// TwinCAT 3 PLC project LoggingExample
// ProgramVersion: 3.1.4024.0
// libraries:
//   Core, 0.0.1.0 (Ziga)
//   Logging, 0.0.1.5 (Ziga)
//   Tc2_Standard, * (Beckhoff Automation GmbH)
//   Tc2_System, * (Beckhoff Automation GmbH)
//   Tc3_Module, * (Beckhoff Automation GmbH)
//   TcError, 0.2.2.0 (Roald87)
//   TcUnit, 1.3.1 (www.tcunit.org)
// project tree:
//   DUTs/ E_SimulationState.TcDUT
//   GVLs/ GVL.TcGVL
//   / PlcTask.TcTTO
//   POUs/ MAIN.TcPOU
//   POUs/Position observer/ FB_PositionObserver_LoggerWithDependencyInjection.TcPOU, FB_PositionObserver_OptionalLoggerWithDependencyInjection.TcPOU, FB_PositionSensorObserverBase.TcPOU
// real-time tasks:
//   TASK PlcTask: cycle T#10ms, priority 20, ADS port 350

CONFIGURATION LoggingExample
    RESOURCE PLC ON TwinCAT3
        TASK PlcTask(INTERVAL := T#10ms, PRIORITY := 20);
        PROGRAM MAIN WITH PlcTask : MAIN;
    END_RESOURCE
END_CONFIGURATION

// ---- DUTs/E_SimulationState.TcDUT
{attribute 'qualified_only'}
{attribute 'strict'}

// Adding this attribute allows to call TO_STRING(enumVariable), which will result in the name of the enum member
{attribute 'to_string'}

TYPE E_SimulationState :
(
	IDLE, 
	BOTTOM, 
	BOTTOM_FOR_10_SECONDS, 
	TOP, TOP_FOR_10_SECONDS 
):= IDLE;
END_TYPE

// ---- GVLs/GVL.TcGVL
{attribute 'qualified_only'}
VAR_GLOBAL
	Logger	: ZigaLibs_Logging.FB_Logger;
	ILogger	: ZigaLibs_Core.I_LoggerEx := Logger;
END_VAR

// ---- POUs/MAIN.TcPOU
PROGRAM MAIN
VAR
	// Instantiating the function block with logger via dependency injection.
	fbPositionObserver_WithLogger : 
		FB_PositionObserver_LoggerWithDependencyInjection(logger := GVL.Logger);
		
	// Instantiating the function block with provided optional logger via dependency injection.
	// For this to work, we need to provide the interface (pointer), instead of the instantiating function block.	
	fbPositionObserver_OptionalLogger_WithLogger : 
		FB_PositionObserver_OptionalLoggerWithDependencyInjection(logger := GVL.ILogger);
		
	// Instantiating the function block without logger via dependency injection.	
	fbPositionObserver_OptionalLogger_WithoutLogger : 
		FB_PositionObserver_OptionalLoggerWithDependencyInjection(logger := 0);
	
		
	eSimulationState			: E_SimulationState := E_SimulationState.IDLE;
	tonPositionTimer			: Tc2_Standard.TON();
	
	
	// Run the simulation
	SIMULATION_RUN				: BOOL;
	observer_simulationState	: ZigaLibs_Core.BoolEx := (variable := SIMULATION_RUN);
	sb							: ZigaLibs_Core.FB_StringBuilder;
	
	firstExecutionAndLoggerValid	: BOOL := TRUE;
END_VAR

VAR CONSTANT
	MY_TARGET_DEVICE_NET_ID 		: Tc2_System.T_AmsNetIdArr := [192,168,56,1,1,1]; // Empty = local
	MY_LOGGER_EXAMPLE_FILE_LOCATION	: Tc2_System.T_MaxString := 'C:\';
	MY_LOGGER_EXAMPLE_FILE_NAME		: Tc2_System.T_MaxString := 'ExampleLog';
END_VAR

// Configure logger
GVL.Logger.AmsAddress.netId := MY_TARGET_DEVICE_NET_ID; 
GVL.Logger.FileProperties.FileLocation := MY_LOGGER_EXAMPLE_FILE_LOCATION;
GVL.Logger.FileProperties.FileName := MY_LOGGER_EXAMPLE_FILE_NAME;

// Logger body still needs to be called
GVL.Logger();

IF GVL.Logger.Ready THEN
	IF firstExecutionAndLoggerValid THEN
		GVL.Logger.LogDefault('====================== FIRST PLC CYCLE EXECUTED ======================');
	END_IF
	firstExecutionAndLoggerValid := FALSE;
	
	// Start/stop simulation logging
	observer_simulationState();
	IF observer_simulationState.HasRisingEdge THEN
		GVL.Logger.LogDefault('====================== STARTING SIMULATION =============================');
		eSimulationState := E_SimulationState.IDLE;
	ELSIF observer_simulationState.HasFallingEdge THEN
		GVL.Logger.LogDefault('====================== STOPPING SIMULATION =============================');
	END_IF
END_IF

// Lets wait for logger to be ready, otherwise date time will be 1970
IF GVL.Logger.Ready AND SIMULATION_RUN THEN		
	// INFO: Check the "Set" implementation for the SimulationState property in MAIN. 
	// You can see state changes being logged in there as well.
	
	// Simulating the positions to generate logs
	CASE SimulationState OF
		E_SimulationState.IDLE:	
			fbPositionObserver_WithLogger.TopPositionSensor := FALSE;
			fbPositionObserver_WithLogger.BottomPositionSensor := FALSE;
			
			fbPositionObserver_OptionalLogger_WithLogger.TopPositionSensor := FALSE;
			fbPositionObserver_OptionalLogger_WithLogger.BottomPositionSensor := FALSE;
			
			fbPositionObserver_OptionalLogger_WithoutLogger.TopPositionSensor := FALSE;
			fbPositionObserver_OptionalLogger_WithoutLogger.BottomPositionSensor := FALSE;
			
			tonPositionTimer(IN := FALSE);
			SimulationState := E_SimulationState.BOTTOM;
			
		E_SimulationState.BOTTOM:
			fbPositionObserver_WithLogger.TopPositionSensor := FALSE;
			fbPositionObserver_WithLogger.BottomPositionSensor := TRUE;
			
			fbPositionObserver_OptionalLogger_WithLogger.TopPositionSensor := FALSE;
			fbPositionObserver_OptionalLogger_WithLogger.BottomPositionSensor := TRUE;
			
			fbPositionObserver_OptionalLogger_WithoutLogger.TopPositionSensor := FALSE;
			fbPositionObserver_OptionalLogger_WithoutLogger.BottomPositionSensor := TRUE;
	
			SimulationState := E_SimulationState.BOTTOM_FOR_10_SECONDS;
			
		E_SimulationState.BOTTOM_FOR_10_SECONDS:
		
			tonPositionTimer(IN := TRUE, PT := T#10S);
			IF tonPositionTimer.Q THEN
				tonPositionTimer(IN := FALSE);
				SimulationState := E_SimulationState.TOP;
			END_IF
			
		E_SimulationState.TOP:
			fbPositionObserver_WithLogger.TopPositionSensor := TRUE;
			fbPositionObserver_WithLogger.BottomPositionSensor := FALSE;
			
			fbPositionObserver_OptionalLogger_WithLogger.TopPositionSensor := TRUE;
			fbPositionObserver_OptionalLogger_WithLogger.BottomPositionSensor := FALSE;
			
			fbPositionObserver_OptionalLogger_WithoutLogger.TopPositionSensor := TRUE;
			fbPositionObserver_OptionalLogger_WithoutLogger.BottomPositionSensor := FALSE;
			
			SimulationState := E_SimulationState.TOP_FOR_10_SECONDS;
			
		E_SimulationState.TOP_FOR_10_SECONDS:
			tonPositionTimer(IN := TRUE, PT := T#10S);
			IF tonPositionTimer.Q THEN
				SimulationState := E_SimulationState.IDLE;
			END_IF
	END_CASE
END_IF


// Call the function blocks here, after simulation
fbPositionObserver_WithLogger();
fbPositionObserver_OptionalLogger_WithLogger();
fbPositionObserver_OptionalLogger_WithoutLogger();

// Gets or sets the simulation state
PROPERTY SimulationState : E_SimulationState
GET
SimulationState := eSimulationState;
END_GET
SET
// Check if value has changed, log the change as well.
IF SimulationState <> eSimulationState THEN
	GVL.Logger.LogDefault(sb.Reset()
		.AddString('========== SIMULATION STATE CHANGED FROM ')
		.AddWithDblQuotationMarks(TO_STRING(eSimulationState))
		.AddString(' TO ')
		.AddWithDblQuotationMarks(TO_STRING(eSimulationState))
		.AddString(' ========== ')
		.Create());
END_IF

eSimulationState := SimulationState;
END_SET
END_PROPERTY

END_PROGRAM

// ---- POUs/Position observer/FB_PositionObserver_LoggerWithDependencyInjection.TcPOU
// A function block with I_LoggerEX as required parameter passed trought FB_Init (dependency injection)
FUNCTION_BLOCK FB_PositionObserver_LoggerWithDependencyInjection EXTENDS FB_PositionSensorObserverBase

// Calling the base class body, FB_PositionSensorObserverBase. It assigns and calls the observers, triggers, ...
// If you want to change how the triggers behave, you could just not call SUPER and do your own implementaiton.
SUPER^();

// =======================================================================================
// ================================ WARNING ==============================================
// =======================================================================================
IF _bottoPositionObserver.HasRisingEdge THEN
	// Lets imagine the bottom position indicates a warning
	_logger.LogWarning(_sb.Reset()
		.AddString('Source: ')
		.AddWithDblQuotationMarks(THIS^.InstanceName)
		.AddString(' Bottom position reached.')
		.Create());
END_IF


// =======================================================================================
// ================================ ERROR ================================================
// =======================================================================================
// And after certain time, we need to trigger an error
IF _bottomPositionError.Q THEN
	_logger.LogError(_sb.Reset()
		.AddString('Source: ').AddWithDblQuotationMarks(THIS^.InstanceName)
		.AddString(' - bottom position has been active for too long!')
		.AddString('Maximum allowed duration is ').AddString(TO_STRING(MAXIMUM_DURATION_AT_BOTTOM_POSITION)).AddString('!')
		.Create());
END_IF

// =======================================================================================
// ================================ INFO =================================================
// =======================================================================================
IF _bottoPositionObserver.HasFallingEdge THEN
	_logger.LogInfo(_sb.Reset()
		.AddString('Source: ').AddWithDblQuotationMarks(THIS^.InstanceName)
		.AddString(' No longer at bottom position. ')
		.AddString('Bottom position was active for ')
		.Create());
END_IF

// =======================================================================================
// ================================ INFO =================================================
// =======================================================================================
IF _topPositionObserver.HasRisingEdge THEN
	_logger.LogInfo(_sb.Reset()
		.AddString('Source: ')
		.AddWithDblQuotationMarks(THIS^.InstanceName)
		.AddString(' Top position reached.')
		.Create());
END_IF

// =======================================================================================
// ================================ INFO =================================================
// =======================================================================================
IF _topPositionObserver.HasFallingEdge THEN
	_logger.LogInfo(_sb.Reset()
		.AddString('Source: ')
		.AddWithDblQuotationMarks(THIS^.InstanceName)
		.AddString(' No longer at top position.')
		.Create());
END_IF

METHOD FB_init : BOOL
VAR_INPUT
	bInitRetains : BOOL; // if TRUE, the retain variables are initialized (warm start / cold start)
	bInCopyCode : BOOL;  // if TRUE, the instance afterwards gets moved into the copy code (online change)
	logger	: ZigaLibs_Core.I_LoggerEx;
END_VAR
// Assign the internal interface to the one provided - interface is basically a pointer. Passing the address this way.
_logger := logger;
END_METHOD

END_FUNCTION_BLOCK

// ---- POUs/Position observer/FB_PositionSensorObserverBase.TcPOU
FUNCTION_BLOCK ABSTRACT FB_PositionSensorObserverBase EXTENDS ZigaLibs_Core.FB_HasInstanceName

VAR
	_topPositionObserver 	: ZigaLibs_Core.BoolEx;
	_topPositionError		: Tc2_Standard.R_TRIG;
	
	_bottoPositionObserver	: ZigaLibs_Core.BoolEx;
	_bottomPositionError	: Tc2_Standard.R_TRIG;
	
	_logger					: ZigaLibs_Core.I_LoggerEx;
	_sb						: ZigaLibs_Core.FB_StringBuilder;
END_VAR

VAR
	{attribute 'hide'}
	_topPositionSensor		: BOOL;
	{attribute 'hide'}
	_bottomPositionSensor	: BOOL;
END_VAR

VAR CONSTANT
	MAXIMUM_DURATION_AT_BOTTOM_POSITION : TIME := T#10S;
	MAXIMUM_DURATION_AT_TOP_POSITION 	: TIME := T#10S;
END_VAR

_topPositionObserver(variable := TopPositionSensor);
_bottoPositionObserver(variable := BottomPositionSensor);
_topPositionError(CLK := _topPositionObserver.HasBeenTrueForAtLeast(MAXIMUM_DURATION_AT_TOP_POSITION));
_bottomPositionError(CLK := _bottoPositionObserver.HasBeenTrueForAtLeast(MAXIMUM_DURATION_AT_BOTTOM_POSITION));

PROPERTY BottomPositionSensor : REFERENCE TO BOOL
GET
BottomPositionSensor REF= _bottomPositionSensor;
END_GET
SET
_bottomPositionSensor := BottomPositionSensor;
END_SET
END_PROPERTY

PROPERTY TopPositionSensor : REFERENCE TO BOOL
GET
TopPositionSensor REF= _topPositionSensor;
END_GET
SET
_topPositionSensor := TopPositionSensor;
END_SET
END_PROPERTY

END_FUNCTION_BLOCK

// ---- POUs/Position observer/FB_PositionObserver_OptionalLoggerWithDependencyInjection.TcPOU
// A function block with I_LoggerEX as an optional parameter passed trought FB_Init (dependency injection)
// This way we can kind of achieve multiple constructors, like in other OOP - the only difference is, we make parameters optional 
FUNCTION_BLOCK FB_PositionObserver_OptionalLoggerWithDependencyInjection EXTENDS FB_PositionSensorObserverBase

// Calling the base class body, FB_PositionSensorObserverBase. It assigns and calls the observers, triggers, ...
// If you want to change how the triggers behave, you could just not call SUPER and do your own implementaiton.
SUPER^();

// Since the interface might not be assigned, we need to check for validity of the pointer.
IF _logger <> 0 THEN
	IF _bottoPositionObserver.HasRisingEdge THEN
		_logger.LogInfo(_sb.Reset()
			.AddString('Source: ')
			.AddWithDblQuotationMarks(THIS^.InstanceName)
			.AddString(' Bottom position reached.')
			.Create());
	END_IF
	
	IF _bottoPositionObserver.HasFallingEdge THEN
		_logger.LogInfo(_sb.Reset()
			.AddString('Source: ')
			.AddWithDblQuotationMarks(THIS^.InstanceName)
			.AddString(' No longer at bottom position.')
			.Create());
	END_IF
	
	IF _topPositionObserver.HasRisingEdge THEN
		_logger.LogInfo(_sb.Reset()
			.AddString('Source: ')
			.AddWithDblQuotationMarks(THIS^.InstanceName)
			.AddString(' Top position reached.')
			.Create());
	END_IF
	
	IF _topPositionObserver.HasFallingEdge THEN
		_logger.LogInfo(_sb.Reset()
			.AddString('Source: ')
			.AddWithDblQuotationMarks(THIS^.InstanceName)
			.AddString(' No longer at top position.')
			.Create());
	END_IF
END_IF

METHOD FB_init : BOOL
VAR_INPUT
	bInitRetains 	: BOOL; // if TRUE, the retain variables are initialized (warm start / cold start)
	bInCopyCode 	: BOOL;  // if TRUE, the instance afterwards gets moved into the copy code (online change)
	logger			: REFERENCE TO ZigaLibs_Core.I_LoggerEx;
END_VAR
// Assign the internal interface to the one provided - interface is basically a pointer. Passing the address this way.
// The difference here is, we are passing a reference to the logger. This means it is optional.
// The user could contruct the fb like this fbSensor : FB_Logger(0); 
// => it is up to us to check the local instance of the _logger
IF __ISVALIDREF(logger) THEN
	_logger := logger;
END_IF
END_METHOD

END_FUNCTION_BLOCK
